TYPE Machine2Machine :
STRUCT
END_STRUCT
END_TYPE

(* stored: Version 1.1.0.1, ProductVersion 3.1.4024.9
   DUT Machine2Machine: Id {2616fa57-c2f1-42db-9109-d2465698e167} *)
